// TIA Portal project "SCDW_TEST_b60eb3d7" (V17)

(* hardware
DEVICE "SCDW_ALARM_PLC"  S7-1200 Station
   slot 0: "Rack_0"  S7-1200 Rack  Rack  V1.0
   slot 1: "SCDW_ALARM_PLC"  CPU 1214C AC/DC/Rly  6ES7 214-1BG40-0XB0  V4.4
*)

// ===== PLC "SCDW_ALARM_PLC"  CPU 1214C AC/DC/Rly =====

VAR_GLOBAL   // PLC tag table "SCDW_ALARM_TAGS"
   "故障反馈1" AT %I0.1 : Bool;
   "故障反馈2" AT %I0.4 : Bool;
   "故障反馈3" AT %I0.7 : Bool;
   "故障反馈4" AT %I1.2 : Bool;
   "故障反馈5" AT %I1.5 : Bool;
   "故障反馈6" AT %I2.2 : Bool;
   "故障反馈7" AT %I2.5 : Bool;
   "蜂鸣器" AT %Q4.7 : Bool;
END_VAR

DATA_BLOCK "内部数据"   // DB1
{ S7_Optimized_Access := 'TRUE' }
VERSION : 0.1
   VAR
      报警脉冲 : Bool;
   END_VAR
BEGIN
END_DATA_BLOCK

FUNCTION "FC_BurnerAlarmRegression" : Void   // FC1, LAD
{ S7_Optimized_Access := 'TRUE' }
   VAR_TEMP   // added for the SCL form of the ladder/FBD networks
      _w1 : Bool;
      _w2 : Bool;
   END_VAR
BEGIN

REGION Network 1: 烧嘴故障上升沿报警
   // 七路故障反馈经O汇合和PBox上升沿检测后置位蜂鸣器。
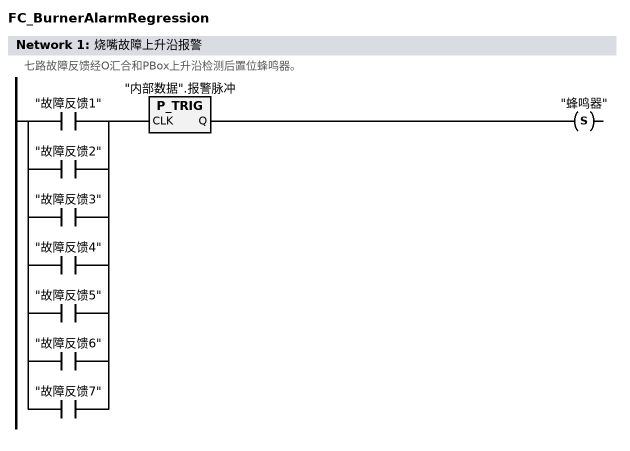
   RUNG wire#powerrail
      Contact( "故障反馈1" )
      wire#w1
      P_Trig( "内部数据".报警脉冲 )
      S_Coil( "蜂鸣器" )
   END_RUNG
   RUNG wire#powerrail
      Contact( "故障反馈2" )
   END_RUNG wire#w1
   RUNG wire#powerrail
      Contact( "故障反馈3" )
   END_RUNG wire#w1
   RUNG wire#powerrail
      Contact( "故障反馈4" )
   END_RUNG wire#w1
   RUNG wire#powerrail
      Contact( "故障反馈5" )
   END_RUNG wire#w1
   RUNG wire#powerrail
      Contact( "故障反馈6" )
   END_RUNG wire#w1
   RUNG wire#powerrail
      Contact( "故障反馈7" )
   END_RUNG wire#w1
   // the same network as SCL:
   #_w1 := "故障反馈1" OR "故障反馈2" OR "故障反馈3" OR "故障反馈4" OR "故障反馈5" OR "故障反馈6" OR "故障反馈7";
   #_w2 := #_w1 AND NOT "内部数据".报警脉冲;   // rising edge
   "内部数据".报警脉冲 := #_w1;
   IF #_w2 THEN "蜂鸣器" := TRUE; END_IF;
END_REGION
END_FUNCTION

ORGANIZATION_BLOCK "Main"   // OB1, LAD, ProgramCycle
TITLE = "Main Program Sweep (Cycle)"
{ S7_Optimized_Access := 'TRUE' }
VERSION : 0.1
   VAR_INPUT
      Initial_Call : Bool;   // Initial call of this OB
      Remanence : Bool;   // =True, if remanent data are available
   END_VAR
BEGIN
END_ORGANIZATION_BLOCK